FUNCTION F_WORD_ARG : ST_Arg
VAR_INPUT
	wInput : WORD;
END_VAR
VAR
	stArg : ST_Arg;
	sysVar_Info : __SYSTEM.VAR_INFO;
END_VAR

sysVar_Info 	:= __VARINFO(wInput);
stArg.TypeClass := sysVar_Info.TypeClass;
stArg.pValue 	:= 0;
stArg.diSize 	:= SIZEOF(wInput);
stArg.sValue 	:= TO_STRING(wInput); 
F_WORD_ARG := stArg;

END_FUNCTION

(* stored: Version 1.1.0.1, ProductVersion 3.1.4024.4
   POU F_WORD_ARG: Id {ed01a839-5be9-4728-80c1-c92c2dd51e7c}, SpecialFunc None *)
